// TwinCAT 3 PLC project Estructurado
// ProgramVersion: 3.1.4024.0
// libraries:
//   CmpBitmapPool, * (System)
//   Tc2_Standard, * (Beckhoff Automation GmbH)
//   Tc2_System, * (Beckhoff Automation GmbH)
//   Tc3_Module, * (Beckhoff Automation GmbH)
//   VisuDialogs, * (System)
// project tree:
//   / GlobalTextList.TcGTLO, PlcTask.TcTTO, Visualization Manager.TcVMO (not stored)
//   POUs/Estacion/ FB_Coordinador_SFC.TcPOU, FB_Estacion.TcPOU
//   POUs/ MAIN.TcPOU
//   POUs/Reloj/ FB_Clock.TcPOU
//   POUs/Tareas/ FB_AlimentadorVerificadorDesplazador_SFC.TcPOU, FB_CheckMaterial_SFC.TcPOU, FB_Descargador_SFC.TcPOU, FB_Rechazador_SFC.TcPOU, FB_ResetDescargador_SFC.TcPOU, FB_SituarPale_SFC.TcPOU, FB_TransferirPale_SFC.TcPOU
//   VISUs/ ImagePool.TcIPO (not stored), Visualization.TcVIS
// (motion and I/O tree: see PLC project manual)
// real-time tasks:
//   TASK PlcTask: cycle T#10ms, priority 20, ADS port 350
//   TASK PlcTask1: cycle T#10ms, priority 21, ADS port 351
// variable links:

CONFIGURATION Estructurado
    RESOURCE PLC ON TwinCAT3
        TASK PlcTask(INTERVAL := T#10ms, PRIORITY := 20);
        PROGRAM MAIN WITH PlcTask : MAIN;
    END_RESOURCE
END_CONFIGURATION

// ---- POUs/MAIN.TcPOU
PROGRAM MAIN
VAR
	
	//Pulsador AT %I*: BOOL;
	//Lampara AT %Q*: BOOL;
	
	Estacion: FB_Estacion;

END_VAR

Estacion();

END_PROGRAM

// ---- POUs/Estacion/FB_Estacion.TcPOU
FUNCTION_BLOCK FB_Estacion
VAR_INPUT
    EstadoPausa: BOOL;
    EstadoReinicia: BOOL;
    CiclosSolicitados: UINT := 0;
	CiclosRechazados: UINT := 0;
    
    Tcheck: TIME := T#1S;
    Treset: TIME := T#1S;
    Tdesplazador: TIME := T#1S;
	Tcinta: TIME := T#0.5S;
END_VAR
VAR_OUTPUT
    CondicionInicial: BOOL := TRUE;
    CiclosPendientes: UINT;
    CiclosAceptados: UINT;
    PaleCodigo: BYTE;
	pieza_ok: BOOL;
    
    // Entradas comunes
	Base_en_alimentador AT %I*: BOOL;
    Pulsador_parada_emergencia AT %I*: BOOL;
    Selector_modo_manual AT %I*: BOOL;
    Pulsador_marcha AT %I*: BOOL;
    Pulsador_parada_NC AT %I*: BOOL := TRUE; // Contacto normalmente cerrado
    EstacionConectada AT %I*: BOOL := TRUE;
    Detector_presion AT %I*: BOOL := TRUE;

    Presencia_pale AT %I*: BOOL;
    Codigo_pale_bit_0 AT %I*: BOOL; //no lo usamos
    Codigo_pale_bit_1 AT %I*: BOOL; //no lo usamos
    Codigo_pale_bit_2 AT %I*: BOOL; //no lo usamos

    // Entradas espeficicas
    //Terminal 6
	Horizontal_descargador_detras AT %I*: BOOL;
	Horizontal_descargador_delante AT %I*: BOOL;
	Vertical_descargador_arriba AT %I*: BOOL;
	Vertical_descargador_abajo AT %I*: BOOL;
	Verificador_arriba AT %I*: BOOL;
	Verificador_abajo AT %I*: BOOL;
	Desplazador_detras AT %I*: BOOL;
	Desplazador_delante AT %I*: BOOL;
	Alimentador_detras AT %I*: BOOL;
	
	
	//Terminal 7
	Alimentador_delante AT %I*: BOOL;
	Vacio_obtenido_vacuostato_descargador AT %I*: BOOL;

END_VAR
VAR
    // Bloques funcionales
    Coordinador: FB_Coordinador_SFC;
	ChequeaMaterial: FB_CheckMaterial_SFC;
	AlimentadorVerificadorDesplazador: FB_AlimentadorVerificadorDesplazador_SFC;
    SituarPale: FB_SituarPale_SFC;
	ResetDescargador: FB_ResetDescargador_SFC;
    Descargador: FB_Descargador_SFC;
    Rechazador: FB_Rechazador_SFC;
    TransferirPale: FB_TransferirPale_SFC;
    
    // Salidas comunes
    Desconecta_parte_operativa AT %Q*: BOOL;
    Lampara_falta_material AT %Q*: BOOL;
    Lampara_marcha AT %Q*: BOOL;
    Lampara_alarma AT %Q*: BOOL;

    Activa_marcha_motor_cinta AT %Q*: BOOL;
    Invierte_marcha_motor_cinta AT %Q*: BOOL;
    Retenedor_pale_baja AT %Q*: BOOL;
    Separador_pale_sube AT %Q*: BOOL;
    
    //Terminal 8
	Descargador_adelante AT %Q*: BOOL;
	Descargador_atras AT %Q*: BOOL;
	Descargador_baja AT %Q*: BOOL;
	Rechazador_adelante AT %Q*: BOOL;
	Verificador_baja AT %Q*: BOOL;
	Desplazador_adelante AT %Q*: BOOL;
	Alimentador_adelante AT %Q*: BOOL;
	Eyector_succiona AT %Q*: BOOL;
END_VAR

// Modo Automático
IF NOT Selector_Modo_Manual THEN
	
	// Bloques Funcionales
	Coordinador(
		CiclosRechazados := CiclosRechazados,
		CiclosPendientes := CiclosPendientes,
		CiclosAceptados := CiclosAceptados,
		CiclosSolicitados := CiclosSolicitados,
		SFCPause := NOT EstadoReinicia AND EstadoPausa,
        SFCReset := EstadoReinicia,
		Ack := TRUE,
        Execute := Pulsador_marcha AND (CiclosSolicitados > 0),
		PaleSituado := SituarPale.Done,
		HayMaterial := ChequeaMaterial.Done,
		Verificado := AlimentadorVerificadorDesplazador.Done,
		DescargadorReseteado := ResetDescargador.Done,
        Rechazado := Rechazador.Done,
		BaseCargada := Descargador.Done,
		PaleTransferido := TransferirPale.Done,
		Base_en_alimentador := Base_en_alimentador,
		pieza_ok := pieza_ok
		
	);
	
	SituarPale(

		SFCPause := NOT EstadoReinicia AND EstadoPausa,
        SFCReset := EstadoReinicia,
        Ack := NOT Coordinador.SituaPale,
        Execute := Coordinador.SituaPale,
        Tcinta := Tcinta,
        Presencia_pale := Presencia_pale,
       	//Codigo_pale_bit_0 := Codigo_pale_bit_0,
        //Codigo_pale_bit_1 := Codigo_pale_bit_1,
        //Codigo_pale_bit_2 := Codigo_pale_bit_2

	);
	
	ChequeaMaterial(
		Ack := NOT Coordinador.ChequeaMaterial,
		SFCPause := NOT EstadoReinicia AND EstadoPausa,
        SFCReset := EstadoReinicia,
		Execute := Coordinador.ChequeaMaterial,
		Base_en_Alimentador := Base_en_alimentador,
		Pulsador_marcha := Pulsador_marcha
	);
	
	AlimentadorVerificadorDesplazador(
		
		Ack := NOT Coordinador.VerificaBase,
		Tcheck := Tcheck,
		SFCPause := NOT EstadoReinicia AND EstadoPausa,
        SFCReset := EstadoReinicia,
		Execute := Coordinador.VerificaBase,
		Alimentador_delante := Alimentador_delante,
		Alimentador_detras := Alimentador_detras,
		Verificador_arriba := Verificador_arriba ,
		Verificador_abajo := Verificador_abajo,
		Desplazador_delante := Desplazador_delante,
		Desplazador_detras := Desplazador_detras, 
		
	);
	
	ResetDescargador(

		Ack := NOT Coordinador.ResetDescargador,
		SFCPause := NOT EstadoReinicia AND EstadoPausa,
        SFCReset := EstadoReinicia,
		Execute := Coordinador.ResetDescargador,
		Horizontal_descargador_detras := Horizontal_descargador_detras,
		Vertical_descargador_arriba := Vertical_descargador_arriba
	);
	
	Descargador(
		
		Ack := NOT Coordinador.CargaBase,
		SFCPause := NOT EstadoReinicia AND EstadoPausa,
        SFCReset := EstadoReinicia,
		Execute := Coordinador.CargaBase,
		Horizontal_descargador_detras := Horizontal_descargador_detras,
		Vertical_descargador_abajo := Vertical_descargador_abajo,
		Vacio_obtenido_vacuostato_descargador := Vacio_obtenido_vacuostato_descargador ,
		Vertical_descargador_arriba := Vertical_descargador_arriba ,
		Horizontal_descargador_delante := Horizontal_descargador_delante ,
	
	);	
		
	Rechazador(
		
		Ack := NOT Coordinador.RechazaBase,
		SFCPause := NOT EstadoReinicia AND EstadoPausa,
        SFCReset := EstadoReinicia,
		Execute := Coordinador.RechazaBase,
		Verificador_abajo := Verificador_abajo
		
	);
	
	TransferirPale(
	
		Ack := NOT Coordinador.TransfierePale,
		SFCPause := NOT EstadoReinicia AND EstadoPausa,
        SFCReset := EstadoReinicia,
		Execute := Coordinador.TransfierePale,

	);
	
	//Acciones Comunes
	Lampara_falta_material := Coordinador.Lampara_falta_material;
	Activa_marcha_motor_cinta := SituarPale.Activa_marcha_motor_cinta OR TransferirPale.Activa_marcha_motor_cinta;
	//CheckMaterial
	Lampara_alarma := ChequeaMaterial.LamparaAlarma;
	Lampara_falta_material := ChequeaMaterial.Lampara_falta_material;
	//TranferirPale
	 Retenedor_pale_baja := TransferirPale.Retenedor_pale_baja;
	 Separador_pale_sube := TransferirPale.Separador_pale_sube;
	//AlimentadorVerificadorDesplazador
	Alimentador_adelante := AlimentadorVerificadorDesplazador.Alimentador_adelante;
	Verificador_baja := AlimentadorVerificadorDesplazador.Verificador_baja;
	Desplazador_adelante := AlimentadorVerificadorDesplazador.Desplazador_adelante;
	pieza_ok := AlimentadorVerificadorDesplazador.pieza_ok;
	//Descargador
	Eyector_succiona := Descargador.Eyector_succiona;
	Descargador_adelante := Descargador.Descargador_adelante;
	Descargador_atras := Descargador.Descargador_atras OR ResetDescargador.Descargador_atras;
	Descargador_baja := Descargador.Descargador_baja;
	//Rechazador
	Rechazador_adelante := Rechazador.Rechazador_adelante;
	
	IF NOT EstadoPausa THEN
	
		EstadoPausa := not Pulsador_parada_NC;
	
	ELSE
	
		EstadoPausa := NOT Pulsador_marcha;
	
	END_IF

END_IF

END_FUNCTION_BLOCK

// ---- POUs/Estacion/FB_Coordinador_SFC.TcPOU
FUNCTION_BLOCK FB_Coordinador_SFC

VAR_IN_OUT
	CiclosPendientes: UINT;
	CiclosAceptados: UINT;
	CiclosRechazados: UINT;
END_VAR
VAR_INPUT
	// SFC-Flags
    SFCPause: BOOL;
    SFCReset: BOOL;
    
    // Indicadores de sincronizacion
    Ack: BOOL := TRUE; //evita que la tarea se realice dos veces
    Execute: BOOL; 
    
    // Parametros de sincronizacion
    PaleSituado: BOOL;
	HayMaterial: BOOL;
    Verificado: BOOL;
	Rechazado: BOOL;
	DescargadorReseteado: BOOL;
    BaseCargada: BOOL;
    PaleTransferido: BOOL;
    
    // Parametros
    CondicionInicial: BOOL;
    CiclosSolicitados: UINT;
	
	//Entradas
	Base_en_Alimentador: BOOL;
	pieza_ok: BOOL;
END_VAR
VAR_OUTPUT
	// Indicadores de sincronizacion
    Done: BOOL;
    Ready: BOOL;

    // Parametros de sincronizacion
    SituaPale: BOOL;
	ChequeaMaterial: BOOL;
    VerificaBase: BOOL;
	ResetDescargador: BOOL;
    RechazaBase: BOOL;
	CargaBase: BOOL;
    TransfierePale: BOOL;
    
    // Salidas
    LamparaAlarma: BOOL;
    LamparaMarcha: BOOL;
	Lampara_falta_material: BOOL;
END_VAR
VAR
	// Bloques funcionales
    CLK: FB_Clock;
END_VAR

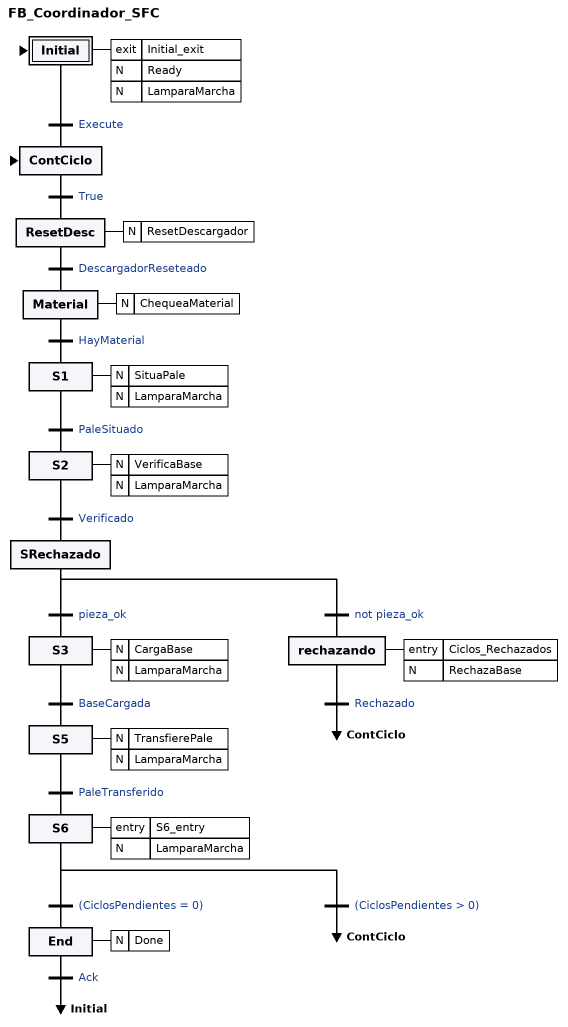
INITIAL_STEP Initial:
    Initial_exit(P0);  // exit action
    Ready(N);
    LamparaMarcha(N);
END_STEP
TRANSITION FROM Initial TO ContCiclo
    := Execute;
END_TRANSITION
STEP ContCiclo:
END_STEP
TRANSITION FROM ContCiclo TO ResetDesc
    := True;
END_TRANSITION
STEP ResetDesc:
    ResetDescargador(N);
END_STEP
TRANSITION FROM ResetDesc TO Material
    := DescargadorReseteado;
END_TRANSITION
STEP Material:
    ChequeaMaterial(N);
END_STEP
TRANSITION FROM Material TO S1
    := HayMaterial;
END_TRANSITION
STEP S1:
    SituaPale(N);
    LamparaMarcha(N);
END_STEP
TRANSITION FROM S1 TO S2
    := PaleSituado;
END_TRANSITION
STEP S2:
    VerificaBase(N);
    LamparaMarcha(N);
END_STEP
TRANSITION FROM S2 TO SRechazado
    := Verificado;
END_TRANSITION
STEP SRechazado:
END_STEP
TRANSITION FROM SRechazado TO S3
    := pieza_ok;
END_TRANSITION
TRANSITION FROM SRechazado TO rechazando
    := not pieza_ok;
END_TRANSITION
STEP rechazando:
    Ciclos_Rechazados(P1);  // entry action
    RechazaBase(N);
END_STEP
TRANSITION FROM rechazando TO ContCiclo
    := Rechazado;
END_TRANSITION
STEP S3:
    CargaBase(N);
    LamparaMarcha(N);
END_STEP
TRANSITION FROM S3 TO S5
    := BaseCargada;
END_TRANSITION
STEP S5:
    TransfierePale(N);
    LamparaMarcha(N);
END_STEP
TRANSITION FROM S5 TO S6
    := PaleTransferido;
END_TRANSITION
STEP S6:
    S6_entry(P1);  // entry action
    LamparaMarcha(N);
END_STEP
TRANSITION FROM S6 TO End
    := (CiclosPendientes = 0);
END_TRANSITION
TRANSITION FROM S6 TO ContCiclo
    := (CiclosPendientes > 0);
END_TRANSITION
STEP End:
    Done(N);
END_STEP
TRANSITION FROM End TO Initial
    := Ack;
END_TRANSITION

ACTION Ciclos_Rechazados:
CiclosRechazados := CiclosRechazados + 1;
END_ACTION

ACTION Initial_exit:
IF (CiclosPendientes = 0) THEN
	CiclosPendientes := CiclosSolicitados;
	CiclosRechazados := 0;
	CiclosAceptados := 0;
END_IF
END_ACTION

ACTION S6_entry:
CiclosPendientes := CiclosPendientes - 1;
CiclosAceptados := CiclosAceptados + 1;
END_ACTION

END_FUNCTION_BLOCK

// ---- POUs/Reloj/FB_Clock.TcPOU
FUNCTION_BLOCK FB_Clock
(*
Square wave oscillator

Copyright (c) 2009-2017 victortorreslopez

GNU General Public License

Version history
2.1, 2017/03/15, VTL: style review (PLCopen Coding Guidelines)
2.0, 2014/12/29, VTL: complete review
1.0, 2009/11/06, VTL: first release
0.0, 2009/11/06, VTL: alfa release
*)
VAR_INPUT
  EN: BOOL := TRUE;	(* ENabled *)
  PT: TIME := T#500ms; (* Semicycle time *)
END_VAR
VAR_OUTPUT
  ET: TIME; (* Elapsed time *)
  Q: BOOL; (* Square wave *)
END_VAR
VAR
  Timer: TON; (* Auto-pilot timer *)
END_VAR

(* OUTPUT FUNCTION *)
IF Timer.Q THEN
  Q := NOT Q;
END_IF

(* FUNCTION BLOCKS *)
Timer(IN := EN AND NOT Timer.Q, PT := PT, ET => ET);

END_FUNCTION_BLOCK

// ---- POUs/Tareas/FB_CheckMaterial_SFC.TcPOU
FUNCTION_BLOCK FB_CheckMaterial_SFC
VAR_INPUT
	// SFC-Flags
    SFCPause: BOOL;
    SFCReset: BOOL;
    
    // Indicadores de sincronizacion
    Ack: BOOL := TRUE; 
    Execute: BOOL;
	
	//Entradas
	Base_en_Alimentador: BOOL;
	Pulsador_marcha: BOOL;
END_VAR
VAR_OUTPUT
	// Indicadores de sincronizacion
    Done: BOOL;
    Ready: BOOL;
	
	//Salidas
	LamparaAlarma: BOOL;
	Lampara_falta_material: BOOL;
END_VAR
VAR
	TMAt: TIME := T#1S;
END_VAR

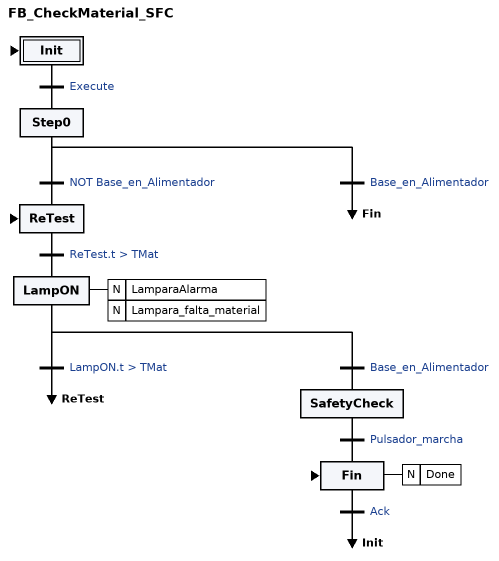
INITIAL_STEP Init:
END_STEP
TRANSITION FROM Init TO Step0
    := Execute;
END_TRANSITION
STEP Step0:
END_STEP
TRANSITION FROM Step0 TO ReTest
    := NOT Base_en_Alimentador;
END_TRANSITION
STEP ReTest:
END_STEP
TRANSITION FROM ReTest TO LampON
    := ReTest.t > TMat;
END_TRANSITION
TRANSITION FROM Step0 TO Fin
    := Base_en_Alimentador;
END_TRANSITION
STEP LampON:
    LamparaAlarma(N);
    Lampara_falta_material(N);
END_STEP
TRANSITION FROM LampON TO ReTest
    := LampON.t > TMat;
END_TRANSITION
TRANSITION FROM LampON TO SafetyCheck
    := Base_en_Alimentador;
END_TRANSITION
STEP SafetyCheck:
END_STEP
TRANSITION FROM SafetyCheck TO Fin
    := Pulsador_marcha;
END_TRANSITION
STEP Fin:
    Done(N);
END_STEP
TRANSITION FROM Fin TO Init
    := Ack;
END_TRANSITION

END_FUNCTION_BLOCK

// ---- POUs/Tareas/FB_AlimentadorVerificadorDesplazador_SFC.TcPOU
FUNCTION_BLOCK FB_AlimentadorVerificadorDesplazador_SFC
VAR_INPUT
	//Tiempo
	Tcheck: TIME := T#1S;
	Tdesplazador: TIME := T#1S;
	
	// SFC-Flags
	SFCPause: BOOL;
	SFCReset: BOOL;
	
	//Indicadores de sincronizacion
	Ack: BOOL:= TRUE;
	Execute: BOOL;
	
	//Entradas
	
	Alimentador_delante: BOOL; //Bajo el verificador
	Alimentador_detras: BOOL;
	Verificador_arriba: BOOL;
	Verificador_abajo: BOOL;
	Desplazador_delante: BOOL;
	Desplazador_detras: BOOL;
	
END_VAR
VAR_OUTPUT
	//indicadores de sincronizacion
	Done: BOOL;
	Ready: BOOL;

	//Salidas
	Alimentador_adelante: BOOL;
	Verificador_baja: BOOL;
	Desplazador_adelante: BOOL;
	
	pieza_ok : BOOL;

END_VAR
VAR
END_VAR

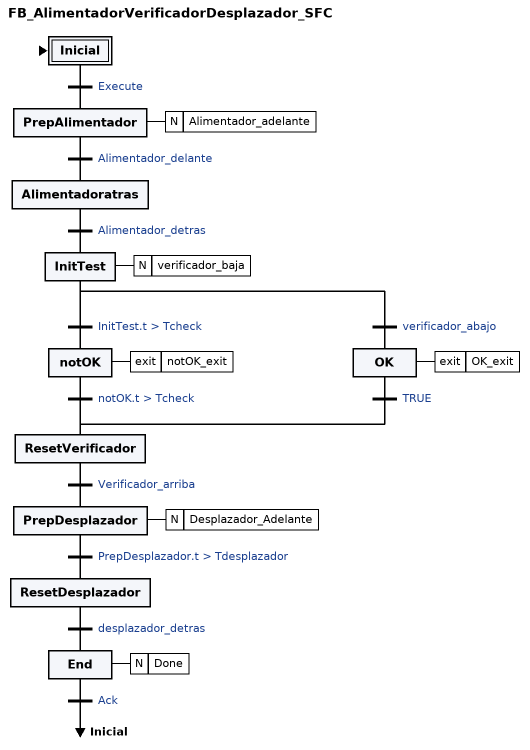
INITIAL_STEP Inicial:
END_STEP
TRANSITION FROM Inicial TO PrepAlimentador
    := Execute;
END_TRANSITION
STEP PrepAlimentador:
    Alimentador_adelante(N);
END_STEP
TRANSITION FROM PrepAlimentador TO Alimentadoratras
    := Alimentador_delante;
END_TRANSITION
STEP Alimentadoratras:
END_STEP
TRANSITION FROM Alimentadoratras TO InitTest
    := Alimentador_detras;
END_TRANSITION
STEP InitTest:
    verificador_baja(N);
END_STEP
TRANSITION FROM InitTest TO notOK
    := InitTest.t > Tcheck;
END_TRANSITION
STEP notOK:
    notOK_exit(P0);  // exit action
END_STEP
TRANSITION FROM notOK TO ResetVerificador
    := notOK.t > Tcheck;
END_TRANSITION
TRANSITION FROM InitTest TO OK
    := verificador_abajo;
END_TRANSITION
STEP OK:
    OK_exit(P0);  // exit action
END_STEP
TRANSITION FROM OK TO ResetVerificador
    := TRUE;
END_TRANSITION
STEP ResetVerificador:
END_STEP
TRANSITION FROM ResetVerificador TO PrepDesplazador
    := Verificador_arriba;
END_TRANSITION
STEP PrepDesplazador:
    Desplazador_Adelante(N);
END_STEP
TRANSITION FROM PrepDesplazador TO ResetDesplazador
    := PrepDesplazador.t > Tdesplazador;
END_TRANSITION
STEP ResetDesplazador:
END_STEP
TRANSITION FROM ResetDesplazador TO End
    := desplazador_detras;
END_TRANSITION
STEP End:
    Done(N);
END_STEP
TRANSITION FROM End TO Inicial
    := Ack;
END_TRANSITION

ACTION notOK_exit:
pieza_ok := FALSE;
END_ACTION

ACTION OK_exit:
pieza_ok := TRUE;
END_ACTION

END_FUNCTION_BLOCK

// ---- POUs/Tareas/FB_SituarPale_SFC.TcPOU
FUNCTION_BLOCK FB_SituarPale_SFC
VAR_INPUT
	//nuestras_variables
	Tcinta: TIME := T#0.5S;

	
    // SFC-Flags
    SFCPause: BOOL;
    SFCReset: BOOL;
    
    // Indicadores de sincronizacion
    Ack: BOOL := TRUE;
    Execute: BOOL;
	
	//Entradas
   	Presencia_pale: BOOL;
	Vertical_descargador_abajo: BOOL;
	Vacio_obtenido_vacuostato_descargador: BOOL;
	Vertical_descargador_arriba: BOOL;
	Horizontal_descargador_delante: BOOL;
	
	
	
END_VAR
VAR_OUTPUT
    // Indicadores de sincronizacion
    Done: BOOL;
    Ready: BOOL;

	//Salidas
	Activa_marcha_motor_cinta: BOOL;
END_VAR
VAR
END_VAR

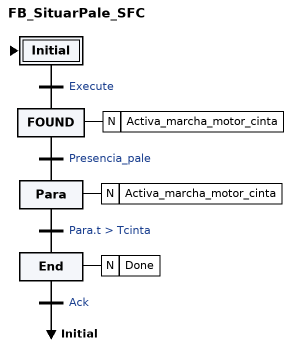
INITIAL_STEP Initial:
END_STEP
TRANSITION FROM Initial TO FOUND
    := Execute;
END_TRANSITION
STEP FOUND:
    Activa_marcha_motor_cinta(N);
END_STEP
TRANSITION FROM FOUND TO Para
    := Presencia_pale;
END_TRANSITION
STEP Para:
    Activa_marcha_motor_cinta(N);
END_STEP
TRANSITION FROM Para TO End
    := Para.t > Tcinta;
END_TRANSITION
STEP End:
    Done(N);
END_STEP
TRANSITION FROM End TO Initial
    := Ack;
END_TRANSITION

END_FUNCTION_BLOCK

// ---- POUs/Tareas/FB_ResetDescargador_SFC.TcPOU
FUNCTION_BLOCK FB_ResetDescargador_SFC

VAR_INPUT
	//nuestras_variables

    // SFC-Flags
    SFCPause: BOOL;
    SFCReset: BOOL;
    
    // Indicadores de sincronizacion
    Ack: BOOL := TRUE;
    Execute: BOOL;
	
	//Entradas
    Horizontal_descargador_detras: BOOL;
	Vertical_descargador_arriba: BOOL;

	
END_VAR
VAR_OUTPUT
    // Indicadores de sincronizacion
    Done: BOOL;
    Ready: BOOL;

	//Salidas
	Descargador_atras: BOOL;
	
END_VAR
VAR
END_VAR

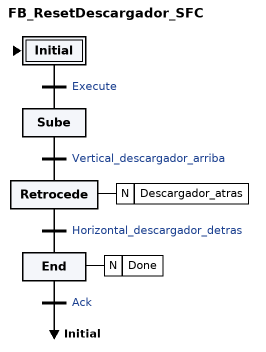
INITIAL_STEP Initial:
END_STEP
TRANSITION FROM Initial TO Sube
    := Execute;
END_TRANSITION
STEP Sube:
END_STEP
TRANSITION FROM Sube TO Retrocede
    := Vertical_descargador_arriba;
END_TRANSITION
STEP Retrocede:
    Descargador_atras(N);
END_STEP
TRANSITION FROM Retrocede TO End
    := Horizontal_descargador_detras;
END_TRANSITION
STEP End:
    Done(N);
END_STEP
TRANSITION FROM End TO Initial
    := Ack;
END_TRANSITION

END_FUNCTION_BLOCK

// ---- POUs/Tareas/FB_Descargador_SFC.TcPOU
FUNCTION_BLOCK FB_Descargador_SFC
VAR_INPUT
	//nuestras_variables
	pieza_ok: BOOL;	

    // SFC-Flags
    SFCPause: BOOL;
    SFCReset: BOOL;
    
    // Indicadores de sincronizacion
    Ack: BOOL := TRUE;
    Execute: BOOL;
	
	//Entradas
    Horizontal_descargador_detras: BOOL;
	Vertical_descargador_abajo: BOOL;
	Vacio_obtenido_vacuostato_descargador: BOOL;
	Vertical_descargador_arriba: BOOL;
	Horizontal_descargador_delante: BOOL;

	
END_VAR
VAR_OUTPUT
    // Indicadores de sincronizacion
    Done: BOOL;
    Ready: BOOL;

	//Salidas
	Descargador_atras: BOOL;
	Descargador_baja: BOOL;
	Eyector_succiona: BOOL;
	Descargador_adelante: BOOL;
END_VAR
VAR
END_VAR

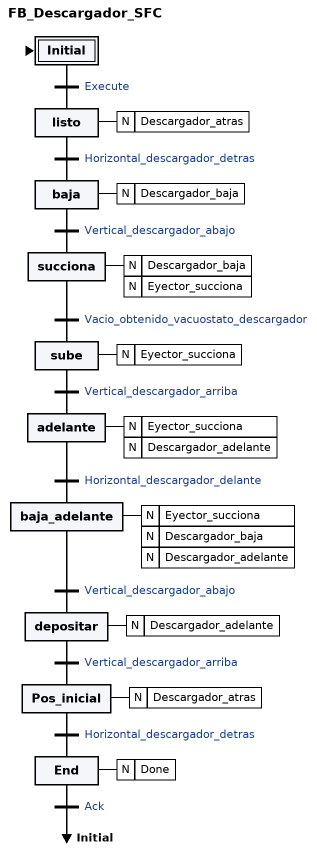
INITIAL_STEP Initial:
END_STEP
TRANSITION FROM Initial TO listo
    := Execute;
END_TRANSITION
STEP listo:
    Descargador_atras(N);
END_STEP
TRANSITION FROM listo TO baja
    := Horizontal_descargador_detras;
END_TRANSITION
STEP baja:
    Descargador_baja(N);
END_STEP
TRANSITION FROM baja TO succiona
    := Vertical_descargador_abajo;
END_TRANSITION
STEP succiona:
    Descargador_baja(N);
    Eyector_succiona(N);
END_STEP
TRANSITION FROM succiona TO sube
    := Vacio_obtenido_vacuostato_descargador;
END_TRANSITION
STEP sube:
    Eyector_succiona(N);
END_STEP
TRANSITION FROM sube TO adelante
    := Vertical_descargador_arriba;
END_TRANSITION
STEP adelante:
    Eyector_succiona(N);
    Descargador_adelante(N);
END_STEP
TRANSITION FROM adelante TO baja_adelante
    := Horizontal_descargador_delante;
END_TRANSITION
STEP baja_adelante:
    Eyector_succiona(N);
    Descargador_baja(N);
    Descargador_adelante(N);
END_STEP
TRANSITION FROM baja_adelante TO depositar
    := Vertical_descargador_abajo;
END_TRANSITION
STEP depositar:
    Descargador_adelante(N);
END_STEP
TRANSITION FROM depositar TO Pos_inicial
    := Vertical_descargador_arriba;
END_TRANSITION
STEP Pos_inicial:
    Descargador_atras(N);
END_STEP
TRANSITION FROM Pos_inicial TO End
    := Horizontal_descargador_detras;
END_TRANSITION
STEP End:
    Done(N);
END_STEP
TRANSITION FROM End TO Initial
    := Ack;
END_TRANSITION

END_FUNCTION_BLOCK

// ---- POUs/Tareas/FB_Rechazador_SFC.TcPOU
FUNCTION_BLOCK FB_Rechazador_SFC
VAR_INPUT
	
	//Tiempo
	Tcheck: TIME := T#1S;	
	
	// SFC-Flags
	SFCPause: BOOL;
	SFCReset: BOOL;
	
	//Indicadores de sincronizacion
	Ack: BOOL:= TRUE;
	Execute: BOOL;
	
	//Entradas
	
	Verificador_abajo: BOOL;

	
END_VAR
VAR_OUTPUT
	//indicadores de sincronizacion
	Done: BOOL;
	Ready: BOOL;

	//Salidas
	Rechazador_adelante: BOOL;
	
END_VAR
VAR
END_VAR

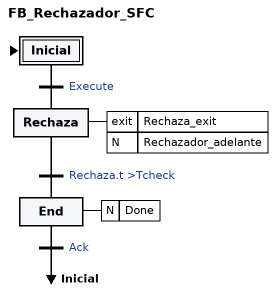
INITIAL_STEP Inicial:
END_STEP
TRANSITION FROM Inicial TO Rechaza
    := Execute;
END_TRANSITION
STEP Rechaza:
    Rechaza_exit(P0);  // exit action
    Rechazador_adelante(N);
END_STEP
TRANSITION FROM Rechaza TO End
    := Rechaza.t >Tcheck;
END_TRANSITION
STEP End:
    Done(N);
END_STEP
TRANSITION FROM End TO Inicial
    := Ack;
END_TRANSITION

ACTION Rechaza_exit:

END_ACTION

END_FUNCTION_BLOCK

// ---- POUs/Tareas/FB_TransferirPale_SFC.TcPOU
FUNCTION_BLOCK FB_TransferirPale_SFC
VAR_INPUT
	
	//Tiempo
	Tcheck: TIME := T#1S;	

	// SFC-Flags
	SFCPause: BOOL;
	SFCReset: BOOL;
	
	//Indicadores de sincronizacion
	Ack: BOOL:= TRUE;
	Execute: BOOL;
	
	//Entradas

	
END_VAR
VAR_OUTPUT
	//indicadores de sincronizacion
	Done: BOOL;
	Ready: BOOL;

	//Salidas
	Retenedor_pale_baja: BOOL;
	Activa_marcha_motor_cinta: BOOL;
	Separador_pale_sube: BOOL;
	
END_VAR
VAR
END_VAR

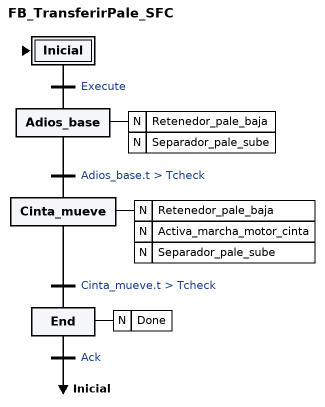
INITIAL_STEP Inicial:
END_STEP
TRANSITION FROM Inicial TO Adios_base
    := Execute;
END_TRANSITION
STEP Adios_base:
    Retenedor_pale_baja(N);
    Separador_pale_sube(N);
END_STEP
TRANSITION FROM Adios_base TO Cinta_mueve
    := Adios_base.t > Tcheck;
END_TRANSITION
STEP Cinta_mueve:
    Retenedor_pale_baja(N);
    Activa_marcha_motor_cinta(N);
    Separador_pale_sube(N);
END_STEP
TRANSITION FROM Cinta_mueve TO End
    := Cinta_mueve.t > Tcheck;
END_TRANSITION
STEP End:
    Done(N);
END_STEP
TRANSITION FROM End TO Inicial
    := Ack;
END_TRANSITION

END_FUNCTION_BLOCK

// ---- GlobalTextList.TcGTLO
TEXTLIST GlobalTextList
  189 = '  ➡ ⬅ ⬇ ⬆ ← → ↓ ↑'
  198 = ' ➙'
  307 = '%i'
  611 = '0'
  472 = '1'
  731 = '<'
  44 = '>'
  12 = 'A+'
  482 = 'A-'
  789 = 'Abajo'
  231 = 'Aceptados'
  66 = 'Alarma'
  224 = 'Alimentador'
  25 = 'Arriba'
  54 = 'Aspirar'
  267 = 'B+'
  782 = 'B-'
  801 = 'C+'
  215 = 'C-'
  701 = 'Ciclos'
  642 = 'Ciclos Completados'
  957 = 'Cinta'
  81 = 'Colocado'
  497 = 'Comenzar'
  143 = 'D+'
  630 = 'D-'
  481 = 'Delante'
  437 = 'Descargador'
  936 = 'Desplazador'
  445 = 'Detrás'
  74 = 'E+'
  781 = 'E-'
  742 = 'E-Stop'
  908 = 'Estado'
  286 = 'Estoy Abajo'
  148 = 'Estoy Arriba'
  955 = 'Eyector'
  417 = 'F+'
  707 = 'F-'
  878 = 'FALTA M.'
  395 = 'FM'
  769 = 'FMS-201                                 ALIMENTADORA DE BASES                                                    VTL     '
  561 = 'Horizontal'
  750 = 'Lámpara'
  45 = 'Marcha'
  634 = 'Material'
  861 = 'Panel'
  463 = 'Parada'
  708 = 'Pausa'
  619 = 'pb'
  935 = 'Pieza NO OK'
  336 = 'Pieza OK'
  741 = 'Pieza Ok'
  524 = 'Planta'
  640 = 'pp'
  783 = 'Preparado'
  330 = 'R+'
  876 = 'Rechazador'
  970 = 'Rechazados'
  888 = 'Rechazads'
  94 = 'Rehczados'
  614 = 'Reset'
  560 = 'Restantes'
  531 = 'Rev'
  452 = 'Run'
  784 = 'S+'
  918 = 'Solicitados'
  815 = 'Succionar'
  643 = 'Tarea'
  710 = 'V+'
  288 = 'V-'
  629 = 'Vacío'
  125 = 'Verificador'
  839 = 'Verificador Activado'
  483 = 'Vertical'
  575 = '➡'
  509 = '⬅'
  381 = '⬆'
  169 = '⬇'
END_TEXTLIST

// ---- VISUs/Visualization.TcVIS
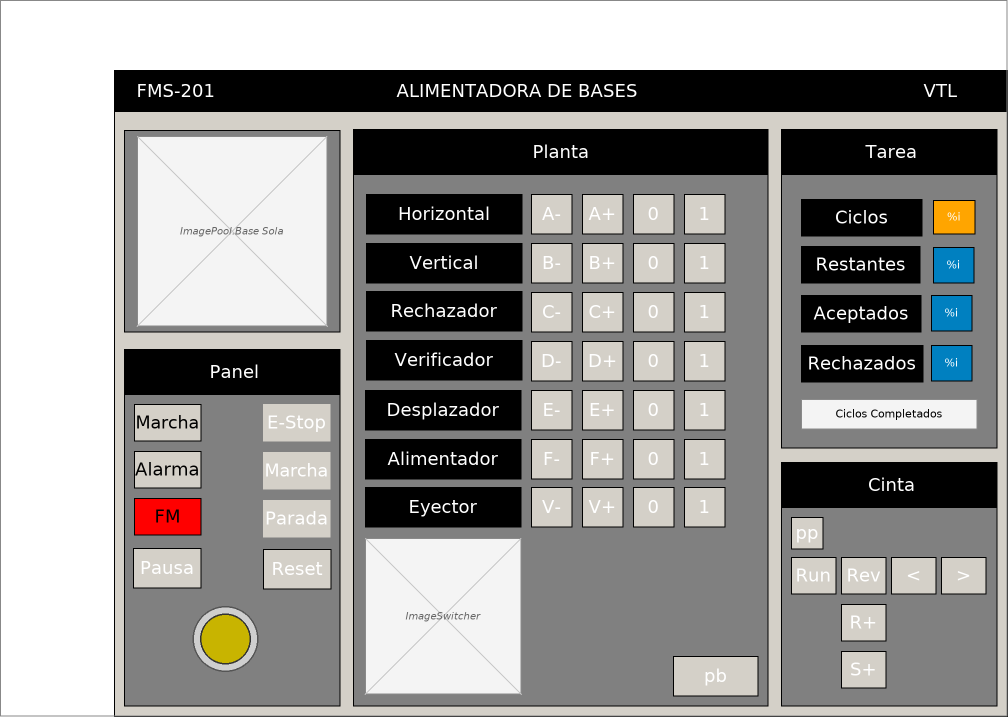
VISUALIZATION Visualization  // 1008x717
    Rectangle (114,111 894x606)
    Rectangle (781,174 216x274)
    Rectangle (353,174 415x532)
    Rectangle (353,129 415x45)
    Label (353,131 416x42), "Planta"
    Rectangle (781,129 216x45)
    Label (831,134 121x36), "Tarea"
    Progressbar (801,399 176x30), "Ciclos Completados", variable: MAIN.test_pieza.Aceptados
    RoundedRectangle (366,194 156x40), "Horizontal"
    Textfield (933,200 42x34), "%i", text variable: MAIN.Estacion.CiclosSolicitados
        OnMouseDown: write MAIN.Estacion.CiclosSolicitados via VisuDialogs.Numpad, min 1, max 10
    RoundedRectangle (801,199 121x37), "Ciclos"
    RoundedRectangle (801,246 119x37), "Restantes"
    RoundedRectangle (801,295 120x37), "Aceptados"
    RoundedRectangle (801,345 122x37), "Rechazados"
    Textfield (933,247 41x36), "%i", text variable: MAIN.Estacion.CiclosPendientes
    Textfield (931,295 41x36), "%i", text variable: MAIN.Estacion.CiclosAceptados
    Textfield (931,345 41x36), "%i", text variable: MAIN.Estacion.CiclosRechazados
    RoundedRectangle (582,243 41x40), "B+", colour toggle: MAIN.Estacion.Descargador_baja
        toggle MAIN.Estacion.Descargador_baja
    Rectangle (781,507 216x199)
    Rectangle (781,462 216x45)
    Label (831,467 121x36), "Cinta"
    Rectangle (124,130 216x202)
    Rectangle (124,394 216x312)
    Rectangle (124,349 216x45)
    Label (174,354 121x36), "Panel"
    Rectangle (114,70 894x41)
    Label (114,71 893x40), "FMS-201 ALIMENTADORA DE BASES VTL"
    RoundedRectangle (366,243 156x40), "Vertical"
    RoundedRectangle (582,194 41x40), "A+", colour toggle: MAIN.Estacion.Descargador_adelante
        tap MAIN.Estacion.Descargador_adelante
    RoundedRectangle (582,292 41x40), "C+", colour toggle: MAIN.Estacion.Rechazador_adelante
        tap MAIN.Estacion.Rechazador_adelante
    RoundedRectangle (582,341 41x40), "D+", colour toggle: MAIN.Estacion.Verificador_baja
        tap MAIN.Estacion.Verificador_baja
    RoundedRectangle (582,390 41x40), "E+", colour toggle: MAIN.Estacion.Desplazador_adelante
        tap MAIN.Estacion.Desplazador_adelante
    RoundedRectangle (582,439 41x40), "F+", colour toggle: MAIN.Estacion.Alimentador_adelante
        tap MAIN.Estacion.Alimentador_adelante
    RoundedRectangle (582,487 41x40), "V+", colour toggle: MAIN.Estacion.Eyector_succiona
        toggle MAIN.Estacion.Eyector_succiona
    RoundedRectangle (366,291 156x40), "Rechazador"
    RoundedRectangle (366,340 156x40), "Verificador"
    RoundedRectangle (365,390 156x40), "Desplazador"
    RoundedRectangle (365,439 156x40), "Alimentador"
    RoundedRectangle (365,487 156x40), "Eyector"
    RoundedRectangle (531,194 41x40), "A-", colour toggle: MAIN.Estacion.Descargador_atras
        tap MAIN.Estacion.Descargador_atras
    RoundedRectangle (633,194 41x40), "0", colour toggle: MAIN.Estacion.Horizontal_descargador_detras
    RoundedRectangle (684,194 41x40), "1", colour toggle: MAIN.Estacion.Horizontal_descargador_delante
    RoundedRectangle (633,243 41x40), "0", colour toggle: MAIN.Estacion.Vertical_descargador_arriba
        tap MAIN.Estacion.Vertical_descargador_arriba
    RoundedRectangle (684,243 41x40), "1", colour toggle: MAIN.Estacion.Vertical_descargador_abajo
        tap MAIN.Estacion.Vertical_descargador_abajo
    RoundedRectangle (633,292 41x40), "0"
    RoundedRectangle (633,341 41x40), "0", colour toggle: MAIN.Estacion.Verificador_arriba
        tap MAIN.Estacion.Verificador_arriba
    RoundedRectangle (633,390 41x40), "0", colour toggle: MAIN.Estacion.Desplazador_detras
        tap MAIN.Estacion.Desplazador_detras
    RoundedRectangle (633,439 41x40), "0", colour toggle: MAIN.Estacion.Alimentador_detras
        tap MAIN.Estacion.Alimentador_detras
    RoundedRectangle (633,487 41x40), "0"
    RoundedRectangle (684,292 41x40), "1"
    RoundedRectangle (684,341 41x40), "1", colour toggle: MAIN.Estacion.Verificador_abajo
        tap MAIN.Estacion.Verificador_abajo
    RoundedRectangle (684,390 41x40), "1"
    RoundedRectangle (684,439 41x40), "1", colour toggle: MAIN.Estacion.Alimentador_delante
        tap MAIN.Estacion.Alimentador_delante
    RoundedRectangle (684,487 41x40), "1", colour toggle: MAIN.Estacion.Vacio_obtenido_vacuostato_descargador
        tap MAIN.Estacion.Vacio_obtenido_vacuostato_descargador
    RoundedRectangle (531,243 41x40), "B-"
    RoundedRectangle (531,292 41x40), "C-"
    RoundedRectangle (531,341 41x40), "D-"
    RoundedRectangle (531,390 41x40), "E-"
    RoundedRectangle (531,439 41x40), "F-"
    RoundedRectangle (531,487 41x40), "V-"
    RoundedRectangle (673,656 85x40), "pb", colour toggle: MAIN.Estacion.Base_en_Alimentador
        tap MAIN.Estacion.Base_en_Alimentador
    RoundedRectangle (134,498 67x37), "FM", colour toggle: MAIN.Estacion.Lampara_falta_material
        tap MAIN.Estacion.Lampara_falta_material
    RoundedRectangle (791,517 32x32), "pp", colour toggle: MAIN.Estacion.Presencia_pale
        tap MAIN.Estacion.Presencia_pale
    RoundedRectangle (941,557 45x37), ">", colour toggle: MAIN.Estacion.Activa_marcha_motor_cinta
        tap MAIN.Estacion.Activa_marcha_motor_cinta
    RoundedRectangle (891,557 45x37), "<", colour toggle: MAIN.Estacion.Invierte_marcha_motor_cinta
        toggle MAIN.Estacion.Invierte_marcha_motor_cinta
    RoundedRectangle (791,557 45x37), "Run", colour toggle: MAIN.Estacion.Activa_marcha_motor_cinta
    RoundedRectangle (841,557 45x37), "Rev", colour toggle: MAIN.Estacion.Invierte_marcha_motor_cinta
    RoundedRectangle (841,604 45x37), "R+", colour toggle: MAIN.Estacion.Retenedor_pale_baja
        toggle MAIN.Estacion.Retenedor_pale_baja
    RoundedRectangle (841,651 45x37), "S+", colour toggle: MAIN.Estacion.Separador_pale_sube
        toggle MAIN.Estacion.Separador_pale_sube
    RoundedRectangle (263,404 67x37), "E-Stop", colour toggle: MAIN.Estacion.Pulsador_parada_emergencia
        tap MAIN.Estacion.Pulsador_parada_emergencia
    RoundedRectangle (263,452 67x37), "Marcha", colour toggle: MAIN.Estacion.Pulsador_marcha
        tap MAIN.Estacion.Pulsador_marcha
    RoundedRectangle (263,500 67x37), "Parada", colour toggle: MAIN.Estacion.Pulsador_parada_NC
        tap MAIN.Estacion.Pulsador_parada_NC
    RoundedRectangle (134,451 67x37), "Alarma", colour toggle: MAIN.Estacion.Lampara_alarma
        tap MAIN.Estacion.Lampara_alarma
    RoundedRectangle (134,404 67x37), "Marcha", colour toggle: MAIN.Estacion.Lampara_marcha
        tap MAIN.Estacion.Lampara_marcha
    Image (137,136 190x190), image: ImagePool.Base Sola
    Lamp1 (187,601 77x76), variable: MAIN.test_pieza.Lampara_falta_material, style: Lamp-Lamp1-Yellow
    ImageSwitcher (365,538 156x156), variable: MAIN.Estacion.pieza_ok, background image: ImagePool.Base OK, image: ImagePool.Base No OK, behaviour: TOGGLE
    RoundedRectangle (133,548 68x40), "Pausa", text variable: MAIN.Estacion.EstadoPausa, colour toggle: MAIN.Estacion.EstadoPausaMAIN.Estacion.EstadoPausa
        tap MAIN.Estacion.EstadoPausa
    RoundedRectangle (263,549 68x40), "Reset", text variable: MAIN.Estacion.EstadoReinicia, colour toggle: MAIN.Estacion.EstadoReinicia
        tap MAIN.Estacion.EstadoReinicia
END_VISUALIZATION
